{attribute 'qualified_only'}
VAR_GLOBAL
	undock: BOOL;
	dock: BOOL;
	cleanin: BOOL;
	cleanout: BOOL;
	piston_moving: BOOL;
	cover_moving: BOOL;
END_VAR

(* stored: Version 1.1.0.1, ProductVersion 3.1.4024.5
   GVL cntrlstate: Id {34f3c4e2-a539-46e2-95c1-633033bf4a94} *)
